(* CODESYS project Acionamento da esteira com dois motores (Set e Reset).project

Project tree, tasks and I/O mapping:
  Device : CODESYS Control Win V3, 3S - Smart Software Solutions GmbH, order no. 305021, version 3.5.11.30
    application Application
      libraries: Standard, * (System)
      task MainTask (cyclic, interval t#20ms, priority 1) calls PLC_PRG
      program PLC_PRG [LD]
      Symbols
*)

// Device/Application/PLC_PRG
PROGRAM PLC_PRG
VAR
	Start: BOOL;
	Stop: BOOL;
	Emergencia: BOOL;
	Esteira_1: BOOL;
	Esteira_2: BOOL;
	Start_Light: BOOL;
	Stop_Light: BOOL;
	Sensor_A: BOOL;
	Sensor_B: BOOL;
	
	
	F_TRIG_0: F_TRIG;
	
	
END_VAR
VAR // added by the converter: edge detectors and wires of the graphical bodies
    _w1, _w2 : BOOL;
END_VAR

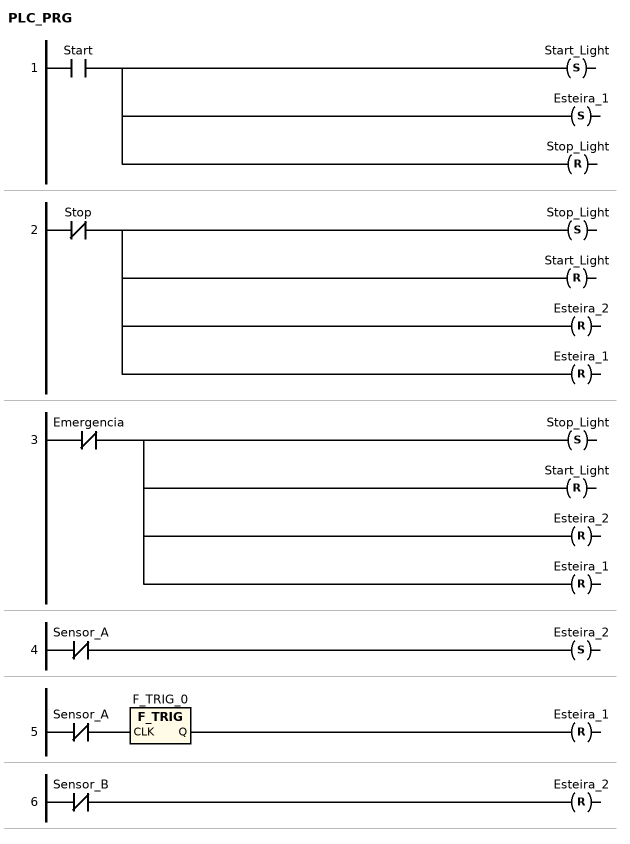
// NETWORK 1
Start_Light S= Start;
Esteira_1 S= Start;
Stop_Light R= Start;

// NETWORK 2
_w1 := NOT Stop;
Stop_Light S= _w1;
Start_Light R= _w1;
Esteira_2 R= _w1;
Esteira_1 R= _w1;

// NETWORK 3
_w2 := NOT Emergencia;
Stop_Light S= _w2;
Start_Light R= _w2;
Esteira_2 R= _w2;
Esteira_1 R= _w2;

// NETWORK 4
Esteira_2 S= NOT Sensor_A;

// NETWORK 5
F_TRIG_0(CLK := NOT Sensor_A); // F_TRIG
Esteira_1 R= F_TRIG_0.Q;

// NETWORK 6
Esteira_2 R= NOT Sensor_B;

END_PROGRAM
